FUNCTION_BLOCK FB_TestStateInitTiming EXTENDS TcUnit.FB_TestSuite
VAR
    stMotionStage: ST_MotionStage;
    fbMotionStageSim: FB_MotionStageSim;
END_VAR

fbMotionStageSim(
    stMotionStage:=stMotionStage,
    nEnableMode:=E_StageEnableMode.DURING_MOTION,
);

PassiveReinit();

METHOD PassiveReinit : BOOL
VAR_INPUT
END_VAR
VAR_INST
    fbStateSetup: FB_StateSetupHelper;
    stDefault: ST_PositionState := (
        fDelta := 0.5,
        fVelocity := 3,
        bMoveOk := TRUE,
        bValid := TRUE
    );
    eEnumSet: UINT;
    eEnumGet: UINT;
    stEpicsToPlc: ST_StateEpicsToPlc;
    stPlcToEpics: ST_StatePlcToEpics;
    fbCore: FB_PositionStateND_Core;
    astMotionStageMax: ARRAY[1..MotionConstants.MAX_STATE_MOTORS] OF ST_MotionStage;
    astPositionStateMax: ARRAY[1..MotionConstants.MAX_STATE_MOTORS] OF ARRAY[1..GeneralConstants.MAX_STATES] OF ST_PositionState;

    mcSetPos: MC_SetPosition;
    nCheckStep: UINT := 0;
    nFurthestStep: UINT;

    nTransitionState: UINT := 99;
    nDoneState: UINT := 99;
    timer: TON;

    nSetPosErrCount: UINT := 0;
    nSetPosErrorID: UDINT;
END_VAR
TEST('PassiveReinit');

// State setup
fbStateSetup(stPositionState:=stDefault, bSetDefault:=TRUE);
fbStateSetup(stPositionState:=astPositionStateMax[1][1], sName:='ONE', fPosition:=10);
fbStateSetup(stPositionState:=astPositionStateMax[1][2], sName:='TWO', fPosition:=20);

// Run the state FB every cycle
astMotionStageMax[1] := stMotionStage;
fbCore(
    astMotionStageMax:=astMotionStageMax,
    astPositionStateMax:=astPositionStateMax,
    stEpicsToPlc:=stEpicsToPlc,
    stPlcToEpics:=stPlcToEpics,
    eEnumSet:=eEnumSet,
    eEnumGet:=eEnumGet,
    bEnable:=TRUE,
    nActiveMotorCount:=1,
);
stMotionStage := astMotionStageMax[1];

// Check and adjust different things as we go
CASE nCheckStep OF
    0:  // State begins at "Unknown", nCurrGoal begins at "Unknown"
        AssertEquals_UINT(
            Expected:=0,
            Actual:=eEnumGet,
            Message:='Did not start in unknown state',
        );
        AssertEquals_UINT(
            Expected:=0,
            Actual:=fbCore.nCurrGoal,
            Message:='Did not start with nCurrGoal unknown',
        );
        mcSetPos(
            Axis:=stMotionStage.Axis,
            Execute:=FALSE,
        );
        nCheckStep := 1;
    1:  // Set the current position to ONE/10
        mcSetPos(
            Axis:=stMotionStage.Axis,
            Execute:=TRUE,
            Position:=10,
        );
        IF mcSetPos.Done THEN
            mcSetPos(
                Axis:=stMotionStage.Axis,
                Execute:=FALSE,
            );
            nCheckStep := 2;
        ELSIF mcSetPos.Error THEN
            nSetPosErrCount := nSetPosErrCount + 1;
            nSetPosErrorID := mcSetPos.ErrorID;
            nCheckStep := 0;
        END_IF
    2:  // Without a move, the state and goal should both change to "ONE" if the position updates
        AssertEquals_UINT(
            Expected:=1,
            Actual:=eEnumGet,
            Message:='Read state did not change to ONE after setpos',
        );
        AssertEquals_UINT(
            Expected:=1,
            Actual:=fbCore.nCurrGoal,
            Message:='nCurrGoal did not change to ONE after setpos',
        );
        // Verify: no move requested
        AssertEquals_LREAL(
            Expected:=0,
            Actual:=stMotionStage.fPosition,
            Delta:=0.001,
            Message:='Set pos routine 1 actually gave us a move!',
        );
        nCheckStep := 3;
    3:  // Same as before, but to 20/TWO
        mcSetPos(
            Axis:=stMotionStage.Axis,
            Execute:=TRUE,
            Position:=20,
        );
        IF mcSetPos.Done THEN
            mcSetPos(
                Axis:=stMotionStage.Axis,
                Execute:=FALSE,
            );
            nCheckStep := 4;
        END_IF
    4:
        AssertEquals_UINT(
            Expected:=2,
            Actual:=eEnumGet,
            Message:='Read state did not change to TWO after setpos',
        );
        AssertEquals_UINT(
            Expected:=2,
            Actual:=fbCore.nCurrGoal,
            Message:='nCurrGoal did not change to TWO after setpos',
        );
        // Verify: no move requested
        AssertEquals_LREAL(
            Expected:=0,
            Actual:=stMotionStage.fPosition,
            Delta:=0.001,
            Message:='Set pos routine 2 actually gave us a move!',
        );
        nCheckStep := 5;
    5:  // Triggering a move should change the goal to the new state, without updating the readback
        eEnumSet := 1;
        nCheckStep := 6;
    6:
        AssertEquals_UINT(
            Expected:=1,
            Actual:=fbCore.nCurrGoal,
            Message:='nCurrGoal did not change to ONE in move',
        );
        // Looking for a readback transition 2 -> 0 -> 1
        // Record the next two transitions
        IF eEnumGet <> 2 AND eEnumGet <> nTransitionState AND eEnumGet <> nDoneState THEN
            nTransitionState := eEnumGet;
        ELSIF eEnumGet <> 2 AND eEnumGet <> nTransitionState THEN
            nDoneState := eEnumGet;
        END_IF
        IF stPlcToEpics.bDone THEN
            AssertEquals_UINT(
                Expected:=0,
                Actual:=nTransitionState,
                Message:='State did not transition 2 -> 0 in move',
            );
            AssertEquals_UINT(
                Expected:=1,
                Actual:=nDoneState,
                Message:='State did not transition 2 -> 0 -> 1 in move',
            );
            nCheckStep := 7;
        END_IF
    7: // The readback and curr goal should match after the move, then end test suite
        AssertEquals_UINT(
            Expected:=1,
            Actual:=eEnumGet,
            Message:='Read state did not change to ONE after move',
        );
        AssertEquals_UINT(
            Expected:=1,
            Actual:=fbCore.nCurrGoal,
            Message:='nCurrGoal did not stay at ONE after move',
        );
        AssertFalse(
            Condition:=timer.Q,
            Message:='Timeout in test',
        );
        TEST_FINISHED();
END_CASE

timer(IN:=TRUE, PT:=T#5s);
IF timer.Q THEN
    nCheckStep := 7;
END_IF
IF nCheckStep < 7 AND nFurthestStep < nCheckStep THEN
    nFurthestStep := nCheckStep;
END_IF
END_METHOD

END_FUNCTION_BLOCK

(* stored: Version 1.1.0.1
   POU FB_TestStateInitTiming: Id {b36fb6c3-2228-4a68-b46d-71d760d78916}, SpecialFunc None
   Method PassiveReinit: Id {f581923a-dba2-4a92-b0c7-df2f67d53bdf} *)
